{attribute 'linkalways'} 
{attribute 'no_explicit_call' := 'This FB is a CLASS and must be accessed using methods or properties'}
{attribute 'enable_dynamic_creation'}
FUNCTION_BLOCK _REAL EXTENDS NumericDatatypeBase
VAR
	localData : REAL;
	activeData : REFERENCE TO REAL REF= localData;
END_VAR

PROPERTY PUBLIC Address : PVOID
GET
Address := ADR(activeData);
END_GET
END_PROPERTY

METHOD PUBLIC ClearReference
VAR_INPUT
END_VAR
activeData REF= localData;
END_METHOD

METHOD PUBLIC Clone : I_Datatype
VAR
    pClone : POINTER TO _REAL;
END_VAR
pClone := __NEW(_REAL(InitialValue := Value));
Clone := pClone^;
END_METHOD

METHOD FB_init : BOOL
VAR_INPUT
	bInitRetains : BOOL; // if TRUE, the retain variables are initialized (warm start / cold start)
	bInCopyCode : BOOL;  // if TRUE, the instance afterwards gets moved into the copy code (online change)
	InitialValue : REAL;
END_VAR
localData := InitialValue;
END_METHOD

PROPERTY PUBLIC IsFloat : BOOL
GET
IsFloat := TRUE;
END_GET
END_PROPERTY

PROPERTY PUBLIC IsSigned : BOOL
GET
IsSigned := TRUE;
END_GET
END_PROPERTY

METHOD PUBLIC MakeReferenceTo
VAR_INPUT
	ReferenceTarget : REFERENCE TO REAL;
END_VAR
activeData REF= ReferenceTarget;
END_METHOD

PROPERTY PUBLIC MaxValue : REAL
GET
MaxValue :=  DatatypeLimits.REAL_MAX_VALUE;
END_GET
END_PROPERTY

PROPERTY PUBLIC MinValue : REAL
GET
MinValue := DatatypeLimits.REAL_MIN_VALUE;
END_GET
END_PROPERTY

METHOD PROTECTED SerializeMaxValue
VAR_INPUT
	Serializer : I_Serializer;
END_VAR
Serializer.AddReal(MaxValue);
END_METHOD

METHOD PROTECTED SerializeMinValue
VAR_INPUT
	Serializer : I_Serializer;
END_VAR
Serializer.AddReal(MinValue);
END_METHOD

METHOD PUBLIC SerializeWith
VAR_INPUT
	Serializer : I_Serializer;
END_VAR
Serializer.AddReal(activeData);
END_METHOD

PROPERTY PUBLIC Size : UDINT
GET
Size := SIZEOF(activeData);
END_GET
END_PROPERTY

METHOD TryDeserializeFrom : BOOL
VAR_INPUT
	Deserializer : I_Deserializer;
	Feedback : I_DeserializerFeedback;
END_VAR
TryDeserializeFrom := Deserializer.TryGetReal(activeData, Feedback);
END_METHOD

METHOD TryMakeReferenceTo : BOOL
VAR_INPUT
	Target : I_Datatype;
END_VAR
VAR
	pTargetData : POINTER TO REAL;
END_VAR
IF NOT (Target.TypeName = TypeName) THEN
	RETURN;
END_IF

pTargetData := Target.Address;
activeData REF= pTargetData^;
TryMakeReferenceTo := TRUE;
END_METHOD

PROPERTY PUBLIC TypeName : T_MAXSTRING
GET
TypeName := 'REAL';
END_GET
END_PROPERTY

PROPERTY PUBLIC Value : REAL
GET
Value := activeData;
END_GET
SET
activeData := Value;
END_SET
END_PROPERTY

END_FUNCTION_BLOCK

(* stored: Version 1.1.0.1, ProductVersion 3.1.4024.12
   POU _REAL: Id {ed8231aa-014c-0b89-0028-924feb4b3de7}, SpecialFunc None
   Folder Constructor: Id {3528773c-d7ad-0b0d-18f2-81143d5de4af}
   Folder Protected: Id {31a44128-d401-4e7f-b5e3-9a64c5cd7486}
   Property Address: Id {d4c0265e-5f37-07e2-1405-56aad7cb6453}
   Get Get: Id {374f109e-e794-030d-0f31-e1b3dba138c9}
   Method ClearReference: Id {18506c58-7109-0bb4-1e46-6d78c59c437e}
   Method Clone: Id {d2ad58e2-cc6a-0e59-1c59-0c3b0e88807d}
   Method FB_init: Id {52e5e737-5c13-094a-1879-7522556f1ed8}
   Property IsFloat: Id {db888af4-7d2e-0761-30e5-93cb9ac46338}
   Get Get: Id {fc1a39e9-9ba0-0ab0-05f9-77163e53fb05}
   Property IsSigned: Id {79e5fc2d-22a4-0f64-0b09-c76fdab6d43d}
   Get Get: Id {d5460f5b-205e-0cba-17f0-3643666a47cc}
   Method MakeReferenceTo: Id {66fc1861-a08b-0f08-3c87-874f7d1c3305}
   Property MaxValue: Id {75b7bc31-5257-49c1-b2f6-9a349776682d}
   Get Get: Id {49a3a31c-5fbf-4a51-9669-c1feec3fac24}
   Property MinValue: Id {7f05c9cc-45eb-40b5-a46b-d0ea831ecedf}
   Get Get: Id {eacb0231-3432-4bdc-a8f5-938266e9d511}
   Method SerializeMaxValue: Id {2323a65c-f9de-479d-81c6-7933b1a717e2}
   Method SerializeMinValue: Id {87ab9796-98b9-434a-bda9-09983c339855}
   Method SerializeWith: Id {5a97850a-1405-02bb-38e6-f44f04b9329e}
   Property Size: Id {27165c67-bd58-0c68-2d5b-c86dce30f1d1}
   Get Get: Id {cc121ac5-c83b-0505-2ad2-83b5a1c0a6fa}
   Method TryDeserializeFrom: Id {69405bb5-13f6-0c0b-0d37-b1e558a29cb5}
   Method TryMakeReferenceTo: Id {37106be5-b9c9-0d3c-1e35-520a6b9d5020}
   Property TypeName: Id {c122af64-7bc0-02cd-1d9e-a1391e87f892}
   Get Get: Id {158e4bad-a707-077e-37a2-700162417ee3}
   Property Value: Id {e0c77763-bd5b-0666-2535-9cf059d74e79}
   Get Get: Id {9836ec7c-9a58-01f9-3cf3-118e937e92dc}
   Set Set: Id {f8018809-8a80-0acd-0204-1847e0a2df21} *)
